{attribute 'qualified_only'}
VAR_GLOBAL
END_VAR

(* stored: Version 1.1.0.1, ProductVersion 3.1.4022.18
   GVL GVL_1: Id {0b3dbaa2-0b98-4911-8405-3cf488d02940} *)
